// TIA Portal V20 export
// export: Created 2026-07-22T09:47:30.5829864Z, ExportSetting WithDefaults, DisplayName Totally Integrated Automation Portal, DisplayVersion V20, DisplayName TIA Portal Openness, DisplayVersion V20, DisplayName TIA Portal Version Control Interface, DisplayVersion V20, DisplayName STEP 7 Professional, DisplayVersion V20, DisplayName STEP 7 Safety, DisplayVersion V20, DisplayName WinCC Basic/Comfort/Advanced, DisplayVersion V20, DisplayName WinCC Professional, DisplayVersion V20, DisplayName WinCC Unified, DisplayVersion V20
FUNCTION_BLOCK "FB_HMI_MIirror"   // FB5, SCL
{ S7_Optimized_Access := 'TRUE' }
VERSION : 0.1
// stored: AutoNumber true, IsIECCheckEnabled false, IsRetainMemResEnabled false, MemoryReserve 100, SetENOAutomatically false, UDAEnableTagReadback false
   VAR
      Lastindex : Int;
   END_VAR
   VAR_TEMP
      idx : Int;
   END_VAR
BEGIN
   // Read selected index and clamp to valid range (1..88)
   #idx := "HMI_Interface_DB".SelectedValveIndex;

   IF #idx < 1 THEN
       #idx := 1;
   ELSIF #idx > 88 THEN
       #idx := 88;
   END_IF;

   // Detect index change -> reset stale commands before mirroring
   IF #idx <> #Lastindex THEN
       "HMI_Interface_DB".OpenCmd := FALSE;
       "HMI_Interface_DB".CloseCmd := FALSE;
       #Lastindex := #idx;
   END_IF;

   // Mirror PLC -> HMI (feedback)
   "HMI_Interface_DB".OpenFB := "Valves_DB".Valve[#idx].OpenFB;
   "HMI_Interface_DB".ClosedFB := "Valves_DB".Valve[#idx].ClosedFB;
   "HMI_Interface_DB".Healthy := "Valves_DB".Valve[#idx].Healthy;
   "HMI_Interface_DB".LocalMode := "Valves_DB".Valve[#idx].LocalMode;

   // Mirror HMI -> PLC (commands)
   "Valves_DB".Valve[#idx].OpenCmd := "HMI_Interface_DB".OpenCmd;
   "Valves_DB".Valve[#idx].CloseCmd := "HMI_Interface_DB".CloseCmd;
END_FUNCTION_BLOCK
